// TIA Portal V20 export
DATA_BLOCK "BK30"   // DB237
// stored: MemoryReserve 100
   VAR
      "SUCTION PAD TOP TAPE VACUUM ON" : Bool := FALSE;
      "SUCTION PAD TOP TAPE VACUUM OFF" : Bool := FALSE;
      "SUCTION PAD BTM TAPE VACUUM ON" : Bool := FALSE;
      "SUCTION PAD BTM TAPE VACUUM OFF" : Bool := FALSE;
      "STACK TABLE V/C ON" : Bool := FALSE;
      "STACK TABLE V/C OFF" : Bool := FALSE;
      SPARE : Bool := FALSE;
      SPARE_1 : Bool := FALSE;
   END_VAR
BEGIN
END_DATA_BLOCK
